Staubli VAL3: Cognex.dtx

bool bCheckRowUpLim = true
bool bDebugProgram = true
bool bDebugSocket
bool bGetID
bool bSafe
bool l_bError
bool resultTrigger = true
camera cCamera[11]
  [0]
    num nErrorCode = 70
    string sErrorMsg[121]
      [0] = "Login> Unrecognized command"
      [1] = "Login> Wrong user name or password"
      [2] = "Login> Communication Error"
      [10] = "Set Online> Command successfull"
      [11] = "Set Online> Unrecognized command"
      [12] = "Set Online> The value given for Int is either out of range, or is not a valid integer"
      [13] = "Set Online> The command could not be executed"
      [14] = "Set Online> Sensor is set Offline manually "
      [15] = "Set Online> User does not have Full Access to execute the command."
      [20] = "Get Online> The In-Sight sensor is currently Offline"
      [21] = "Get Online> The In-Sight sensor is currently Online"
      [30] = "Load File> Command successfull"
      [31] = "Load File> Unrecognized command"
      [32] = "Load File> The filename is missing"
      [33] = "Load File> The job failed to load, the sensor is Online, or the file was not found"
      [34] = "Load File> The job to be loaded was not found, or the sensor is out of memory"
      [35] = "Load File> User does not have Full Access"
      [40] = "get File> Command successfull"
      [41] = "get File> Unrecognized command"
      [42] = "get File> The active job has not been saved"
      [50] = "Save file> Command successfull"
      [51] = "Save file> Unrecognized command"
      [52] = "Save file> The filename is missing"
      [53] = "Save file>The job failed to save, the sensor is Online or the file was not found"
      [54] = "Save file> User does not have Full Access "
      [60] = "Set Event> Command successfull"
      [61] = "Set Event> Unrecognized command"
      [62] = "Set Event> The number is either out of range or not an integer"
      [63] = "Set Event>The command could not be executed, or the sensor is Offline"
      [64] = "Set Event> User does not have Full Access "
      [70] = "Get Value> Command successfull"
      [71] = "Get Value> Unrecognized command"
      [72] = "Get Value> Cell ID is invalid"
      [73] = "Get Value> The command could not be executed"
      [80] = "Set Float> Command successfull"
      [81] = "Set Float> Unrecognized command"
      [82] = "Set Float> Cell ID is invalid, or not a float"
      [83] = "Set Float> Cell was not created by the EditFloat function"
      [84] = "Set Float> User does not have Full Access "
      [90] = "Set Integer> Command successfull"
      [91] = "Set Integer>Unrecognized command"
      [92] = "Set Integer>Cell ID invalid, or not an integer"
      [93] = "Set Integer> Integer value is outside of the control's valid range or cell was not created by the EditInt function"
      [94] = "Set Integer> User does not have Full Access"
      [100] = "Set String> Command successfull"
      [101] = "Set String> Unrecognized command"
      [102] = "Set String> Cell ID invalid"
      [103] = "Set String> String is too longer or the cell does not contain an EditString function"
      [104] = "Set String> User does not have Full Access"
      [110] = "Cell Format> OK"
      [111] = "Cell Format> Invalid column"
      [112] = "Cell Format> Invalid row"
      [113] = "Cell Format> Row number out of range"
    sio sSocket = {link=Socket\sCognex1}
    bool bConnected
  [1]
    num nErrorCode = 70
    string sErrorMsg[120]
      [0] = "Login> Unrecognized command"
      [1] = "Login> Wrong user name or password"
      [2] = "Login> Communication Error"
      [10] = "Set Online> Command successfully"
      [11] = "Set Online> Unrecognized command"
      [12] = "Set Online> The value given for Int is either out of range, or is not a valid integer"
      [13] = "Set Online> The command could not be executed"
      [14] = "Set Online> Sensor is set Offline manually "
      [15] = "Set Online> User does not have Full Access to execute the command."
      [20] = "Get Online> The In-Sight sensor is currently Offline"
      [21] = "Get Online> The In-Sight sensor is currently Online"
      [30] = "Load File> Command successfully"
      [31] = "Load File> Unrecognized command"
      [32] = "Load File> The filename is missing"
      [33] = "Load File> The job failed to load, the sensor is Online, or the file was not found"
      [34] = "Load File> The job to be loaded was not found, or the sensor is out of memory"
      [35] = "Load File> User does not have Full Access"
      [40] = "get File> Command successfully"
      [41] = "get File> Unrecognized command"
      [42] = "get File> The active job has not been saved"
      [50] = "Save file> Command successfully"
      [51] = "Save file> Unrecognized command"
      [52] = "Save file> The filename is missing"
      [53] = "Save file>The job failed to save, the sensor is Online or the file was not found"
      [54] = "Save file> User does not have Full Access "
      [60] = "Set Event> Command successfully"
      [61] = "Set Event> Unrecognized command"
      [62] = "Set Event> The number is either out of range or not an integer"
      [63] = "Set Event>The command could not be executed, or the sensor is Offline"
      [64] = "Set Event> User does not have Full Access "
      [70] = "Get Value> Command successfully"
      [71] = "Get Value> Unrecognized command"
      [72] = "Get Value> Cell ID is invalid"
      [73] = "Get Value> The command could not be executed"
      [80] = "Set Float> Command successfully"
      [81] = "Set Float> Unrecognized command"
      [82] = "Set Float> Cell ID is invalid, or not a float"
      [83] = "Set Float> Cell was not created by the EditFloat function"
      [84] = "Set Float> User does not have Full Access "
      [90] = "Set Integer> Command successfully"
      [91] = "Set Integer>Unrecognized command"
      [92] = "Set Integer>Cell ID invalid, or not an integer"
      [93] = "Set Integer> Integer value is outside of the control's valid range or cell was not created by the EditInt function"
      [94] = "Set Integer> User does not have Full Access"
      [100] = "Set String> Command successfully"
      [101] = "Set String> Unrecognized command"
      [102] = "Set String> Cell ID invalid"
      [103] = "Set String> String is too longer or the cell does not contain an EditString function"
      [104] = "Set String> User does not have Full Access"
      [110] = "Cell Format> OK"
      [111] = "Cell Format> Invalid column"
      [112] = "Cell Format> Invalid row"
      [113] = "Cell Format> Row number out of range"
    sio sSocket = {link=Socket\sCognex1}
    bool bConnected
  [2]
    num nErrorCode
    string sErrorMsg[120]
      [0] = "Login> Unrecognized command"
      [1] = "Login> Wrong user name or password"
      [2] = "Login> Communication Error"
      [10] = "Set Online> Command successfully"
      [11] = "Set Online> Unrecognized command"
      [12] = "Set Online> The value given for Int is either out of range, or is not a valid integer"
      [13] = "Set Online> The command could not be executed"
      [14] = "Set Online> Sensor is set Offline manually "
      [15] = "Set Online> User does not have Full Access to execute the command."
      [20] = "Get Online> The In-Sight sensor is currently Offline"
      [21] = "Get Online> The In-Sight sensor is currently Online"
      [30] = "Load File> Command successfully"
      [31] = "Load File> Unrecognized command"
      [32] = "Load File> The filename is missing"
      [33] = "Load File> The job failed to load, the sensor is Online, or the file was not found"
      [34] = "Load File> The job to be loaded was not found, or the sensor is out of memory"
      [35] = "Load File> User does not have Full Access"
      [40] = "get File> Command successfully"
      [41] = "get File> Unrecognized command"
      [42] = "get File> The active job has not been saved"
      [50] = "Save file> Command successfully"
      [51] = "Save file> Unrecognized command"
      [52] = "Save file> The filename is missing"
      [53] = "Save file>The job failed to save, the sensor is Online or the file was not found"
      [54] = "Save file> User does not have Full Access "
      [60] = "Set Event> Command successfully"
      [61] = "Set Event> Unrecognized command"
      [62] = "Set Event> The number is either out of range or not an integer"
      [63] = "Set Event>The command could not be executed, or the sensor is Offline"
      [64] = "Set Event> User does not have Full Access "
      [70] = "Get Value> Command successfully"
      [71] = "Get Value> Unrecognized command"
      [72] = "Get Value> Cell ID is invalid"
      [73] = "Get Value> The command could not be executed"
      [80] = "Set Float> Command successfully"
      [81] = "Set Float> Unrecognized command"
      [82] = "Set Float> Cell ID is invalid, or not a float"
      [83] = "Set Float> Cell was not created by the EditFloat function"
      [84] = "Set Float> User does not have Full Access "
      [90] = "Set Integer> Command successfully"
      [91] = "Set Integer>Unrecognized command"
      [92] = "Set Integer>Cell ID invalid, or not an integer"
      [93] = "Set Integer> Integer value is outside of the control's valid range or cell was not created by the EditInt function"
      [94] = "Set Integer> User does not have Full Access"
      [100] = "Set String> Command successfully"
      [101] = "Set String> Unrecognized command"
      [102] = "Set String> Cell ID invalid"
      [103] = "Set String> String is too longer or the cell does not contain an EditString function"
      [104] = "Set String> User does not have Full Access"
      [110] = "Cell Format> OK"
      [111] = "Cell Format> Invalid column"
      [112] = "Cell Format> Invalid row"
      [113] = "Cell Format> Row number out of range"
    sio sSocket
    bool bConnected
  [3]
    num nErrorCode
    string sErrorMsg[120]
      [0] = "Login> Unrecognized command"
      [1] = "Login> Wrong user name or password"
      [2] = "Login> Communication Error"
      [10] = "Set Online> Command successfully"
      [11] = "Set Online> Unrecognized command"
      [12] = "Set Online> The value given for Int is either out of range, or is not a valid integer"
      [13] = "Set Online> The command could not be executed"
      [14] = "Set Online> Sensor is set Offline manually "
      [15] = "Set Online> User does not have Full Access to execute the command."
      [20] = "Get Online> The In-Sight sensor is currently Offline"
      [21] = "Get Online> The In-Sight sensor is currently Online"
      [30] = "Load File> Command successfully"
      [31] = "Load File> Unrecognized command"
      [32] = "Load File> The filename is missing"
      [33] = "Load File> The job failed to load, the sensor is Online, or the file was not found"
      [34] = "Load File> The job to be loaded was not found, or the sensor is out of memory"
      [35] = "Load File> User does not have Full Access"
      [40] = "get File> Command successfully"
      [41] = "get File> Unrecognized command"
      [42] = "get File> The active job has not been saved"
      [50] = "Save file> Command successfully"
      [51] = "Save file> Unrecognized command"
      [52] = "Save file> The filename is missing"
      [53] = "Save file>The job failed to save, the sensor is Online or the file was not found"
      [54] = "Save file> User does not have Full Access "
      [60] = "Set Event> Command successfully"
      [61] = "Set Event> Unrecognized command"
      [62] = "Set Event> The number is either out of range or not an integer"
      [63] = "Set Event>The command could not be executed, or the sensor is Offline"
      [64] = "Set Event> User does not have Full Access "
      [70] = "Get Value> Command successfully"
      [71] = "Get Value> Unrecognized command"
      [72] = "Get Value> Cell ID is invalid"
      [73] = "Get Value> The command could not be executed"
      [80] = "Set Float> Command successfully"
      [81] = "Set Float> Unrecognized command"
      [82] = "Set Float> Cell ID is invalid, or not a float"
      [83] = "Set Float> Cell was not created by the EditFloat function"
      [84] = "Set Float> User does not have Full Access "
      [90] = "Set Integer> Command successfully"
      [91] = "Set Integer>Unrecognized command"
      [92] = "Set Integer>Cell ID invalid, or not an integer"
      [93] = "Set Integer> Integer value is outside of the control's valid range or cell was not created by the EditInt function"
      [94] = "Set Integer> User does not have Full Access"
      [100] = "Set String> Command successfully"
      [101] = "Set String> Unrecognized command"
      [102] = "Set String> Cell ID invalid"
      [103] = "Set String> String is too longer or the cell does not contain an EditString function"
      [104] = "Set String> User does not have Full Access"
      [110] = "Cell Format> OK"
      [111] = "Cell Format> Invalid column"
      [112] = "Cell Format> Invalid row"
      [113] = "Cell Format> Row number out of range"
    sio sSocket
    bool bConnected
  [4]
    num nErrorCode
    string sErrorMsg[120]
      [0] = "Login> Unrecognized command"
      [1] = "Login> Wrong user name or password"
      [2] = "Login> Communication Error"
      [10] = "Set Online> Command successfully"
      [11] = "Set Online> Unrecognized command"
      [12] = "Set Online> The value given for Int is either out of range, or is not a valid integer"
      [13] = "Set Online> The command could not be executed"
      [14] = "Set Online> Sensor is set Offline manually "
      [15] = "Set Online> User does not have Full Access to execute the command."
      [20] = "Get Online> The In-Sight sensor is currently Offline"
      [21] = "Get Online> The In-Sight sensor is currently Online"
      [30] = "Load File> Command successfully"
      [31] = "Load File> Unrecognized command"
      [32] = "Load File> The filename is missing"
      [33] = "Load File> The job failed to load, the sensor is Online, or the file was not found"
      [34] = "Load File> The job to be loaded was not found, or the sensor is out of memory"
      [35] = "Load File> User does not have Full Access"
      [40] = "get File> Command successfully"
      [41] = "get File> Unrecognized command"
      [42] = "get File> The active job has not been saved"
      [50] = "Save file> Command successfully"
      [51] = "Save file> Unrecognized command"
      [52] = "Save file> The filename is missing"
      [53] = "Save file>The job failed to save, the sensor is Online or the file was not found"
      [54] = "Save file> User does not have Full Access "
      [60] = "Set Event> Command successfully"
      [61] = "Set Event> Unrecognized command"
      [62] = "Set Event> The number is either out of range or not an integer"
      [63] = "Set Event>The command could not be executed, or the sensor is Offline"
      [64] = "Set Event> User does not have Full Access "
      [70] = "Get Value> Command successfully"
      [71] = "Get Value> Unrecognized command"
      [72] = "Get Value> Cell ID is invalid"
      [73] = "Get Value> The command could not be executed"
      [80] = "Set Float> Command successfully"
      [81] = "Set Float> Unrecognized command"
      [82] = "Set Float> Cell ID is invalid, or not a float"
      [83] = "Set Float> Cell was not created by the EditFloat function"
      [84] = "Set Float> User does not have Full Access "
      [90] = "Set Integer> Command successfully"
      [91] = "Set Integer>Unrecognized command"
      [92] = "Set Integer>Cell ID invalid, or not an integer"
      [93] = "Set Integer> Integer value is outside of the control's valid range or cell was not created by the EditInt function"
      [94] = "Set Integer> User does not have Full Access"
      [100] = "Set String> Command successfully"
      [101] = "Set String> Unrecognized command"
      [102] = "Set String> Cell ID invalid"
      [103] = "Set String> String is too longer or the cell does not contain an EditString function"
      [104] = "Set String> User does not have Full Access"
      [110] = "Cell Format> OK"
      [111] = "Cell Format> Invalid column"
      [112] = "Cell Format> Invalid row"
      [113] = "Cell Format> Row number out of range"
    sio sSocket
    bool bConnected
  [5]
    num nErrorCode
    string sErrorMsg[120]
      [0] = "Login> Unrecognized command"
      [1] = "Login> Wrong user name or password"
      [2] = "Login> Communication Error"
      [10] = "Set Online> Command successfully"
      [11] = "Set Online> Unrecognized command"
      [12] = "Set Online> The value given for Int is either out of range, or is not a valid integer"
      [13] = "Set Online> The command could not be executed"
      [14] = "Set Online> Sensor is set Offline manually "
      [15] = "Set Online> User does not have Full Access to execute the command."
      [20] = "Get Online> The In-Sight sensor is currently Offline"
      [21] = "Get Online> The In-Sight sensor is currently Online"
      [30] = "Load File> Command successfully"
      [31] = "Load File> Unrecognized command"
      [32] = "Load File> The filename is missing"
      [33] = "Load File> The job failed to load, the sensor is Online, or the file was not found"
      [34] = "Load File> The job to be loaded was not found, or the sensor is out of memory"
      [35] = "Load File> User does not have Full Access"
      [40] = "get File> Command successfully"
      [41] = "get File> Unrecognized command"
      [42] = "get File> The active job has not been saved"
      [50] = "Save file> Command successfully"
      [51] = "Save file> Unrecognized command"
      [52] = "Save file> The filename is missing"
      [53] = "Save file>The job failed to save, the sensor is Online or the file was not found"
      [54] = "Save file> User does not have Full Access "
      [60] = "Set Event> Command successfully"
      [61] = "Set Event> Unrecognized command"
      [62] = "Set Event> The number is either out of range or not an integer"
      [63] = "Set Event>The command could not be executed, or the sensor is Offline"
      [64] = "Set Event> User does not have Full Access "
      [70] = "Get Value> Command successfully"
      [71] = "Get Value> Unrecognized command"
      [72] = "Get Value> Cell ID is invalid"
      [73] = "Get Value> The command could not be executed"
      [80] = "Set Float> Command successfully"
      [81] = "Set Float> Unrecognized command"
      [82] = "Set Float> Cell ID is invalid, or not a float"
      [83] = "Set Float> Cell was not created by the EditFloat function"
      [84] = "Set Float> User does not have Full Access "
      [90] = "Set Integer> Command successfully"
      [91] = "Set Integer>Unrecognized command"
      [92] = "Set Integer>Cell ID invalid, or not an integer"
      [93] = "Set Integer> Integer value is outside of the control's valid range or cell was not created by the EditInt function"
      [94] = "Set Integer> User does not have Full Access"
      [100] = "Set String> Command successfully"
      [101] = "Set String> Unrecognized command"
      [102] = "Set String> Cell ID invalid"
      [103] = "Set String> String is too longer or the cell does not contain an EditString function"
      [104] = "Set String> User does not have Full Access"
      [110] = "Cell Format> OK"
      [111] = "Cell Format> Invalid column"
      [112] = "Cell Format> Invalid row"
      [113] = "Cell Format> Row number out of range"
    sio sSocket
    bool bConnected
  [6]
    num nErrorCode
    string sErrorMsg[120]
      [0] = "Login> Unrecognized command"
      [1] = "Login> Wrong user name or password"
      [2] = "Login> Communication Error"
      [10] = "Set Online> Command successfully"
      [11] = "Set Online> Unrecognized command"
      [12] = "Set Online> The value given for Int is either out of range, or is not a valid integer"
      [13] = "Set Online> The command could not be executed"
      [14] = "Set Online> Sensor is set Offline manually "
      [15] = "Set Online> User does not have Full Access to execute the command."
      [20] = "Get Online> The In-Sight sensor is currently Offline"
      [21] = "Get Online> The In-Sight sensor is currently Online"
      [30] = "Load File> Command successfully"
      [31] = "Load File> Unrecognized command"
      [32] = "Load File> The filename is missing"
      [33] = "Load File> The job failed to load, the sensor is Online, or the file was not found"
      [34] = "Load File> The job to be loaded was not found, or the sensor is out of memory"
      [35] = "Load File> User does not have Full Access"
      [40] = "get File> Command successfully"
      [41] = "get File> Unrecognized command"
      [42] = "get File> The active job has not been saved"
      [50] = "Save file> Command successfully"
      [51] = "Save file> Unrecognized command"
      [52] = "Save file> The filename is missing"
      [53] = "Save file>The job failed to save, the sensor is Online or the file was not found"
      [54] = "Save file> User does not have Full Access "
      [60] = "Set Event> Command successfully"
      [61] = "Set Event> Unrecognized command"
      [62] = "Set Event> The number is either out of range or not an integer"
      [63] = "Set Event>The command could not be executed, or the sensor is Offline"
      [64] = "Set Event> User does not have Full Access "
      [70] = "Get Value> Command successfully"
      [71] = "Get Value> Unrecognized command"
      [72] = "Get Value> Cell ID is invalid"
      [73] = "Get Value> The command could not be executed"
      [80] = "Set Float> Command successfully"
      [81] = "Set Float> Unrecognized command"
      [82] = "Set Float> Cell ID is invalid, or not a float"
      [83] = "Set Float> Cell was not created by the EditFloat function"
      [84] = "Set Float> User does not have Full Access "
      [90] = "Set Integer> Command successfully"
      [91] = "Set Integer>Unrecognized command"
      [92] = "Set Integer>Cell ID invalid, or not an integer"
      [93] = "Set Integer> Integer value is outside of the control's valid range or cell was not created by the EditInt function"
      [94] = "Set Integer> User does not have Full Access"
      [100] = "Set String> Command successfully"
      [101] = "Set String> Unrecognized command"
      [102] = "Set String> Cell ID invalid"
      [103] = "Set String> String is too longer or the cell does not contain an EditString function"
      [104] = "Set String> User does not have Full Access"
      [110] = "Cell Format> OK"
      [111] = "Cell Format> Invalid column"
      [112] = "Cell Format> Invalid row"
      [113] = "Cell Format> Row number out of range"
    sio sSocket
    bool bConnected
  [7]
    num nErrorCode
    string sErrorMsg[120]
      [0] = "Login> Unrecognized command"
      [1] = "Login> Wrong user name or password"
      [2] = "Login> Communication Error"
      [10] = "Set Online> Command successfully"
      [11] = "Set Online> Unrecognized command"
      [12] = "Set Online> The value given for Int is either out of range, or is not a valid integer"
      [13] = "Set Online> The command could not be executed"
      [14] = "Set Online> Sensor is set Offline manually "
      [15] = "Set Online> User does not have Full Access to execute the command."
      [20] = "Get Online> The In-Sight sensor is currently Offline"
      [21] = "Get Online> The In-Sight sensor is currently Online"
      [30] = "Load File> Command successfully"
      [31] = "Load File> Unrecognized command"
      [32] = "Load File> The filename is missing"
      [33] = "Load File> The job failed to load, the sensor is Online, or the file was not found"
      [34] = "Load File> The job to be loaded was not found, or the sensor is out of memory"
      [35] = "Load File> User does not have Full Access"
      [40] = "get File> Command successfully"
      [41] = "get File> Unrecognized command"
      [42] = "get File> The active job has not been saved"
      [50] = "Save file> Command successfully"
      [51] = "Save file> Unrecognized command"
      [52] = "Save file> The filename is missing"
      [53] = "Save file>The job failed to save, the sensor is Online or the file was not found"
      [54] = "Save file> User does not have Full Access "
      [60] = "Set Event> Command successfully"
      [61] = "Set Event> Unrecognized command"
      [62] = "Set Event> The number is either out of range or not an integer"
      [63] = "Set Event>The command could not be executed, or the sensor is Offline"
      [64] = "Set Event> User does not have Full Access "
      [70] = "Get Value> Command successfully"
      [71] = "Get Value> Unrecognized command"
      [72] = "Get Value> Cell ID is invalid"
      [73] = "Get Value> The command could not be executed"
      [80] = "Set Float> Command successfully"
      [81] = "Set Float> Unrecognized command"
      [82] = "Set Float> Cell ID is invalid, or not a float"
      [83] = "Set Float> Cell was not created by the EditFloat function"
      [84] = "Set Float> User does not have Full Access "
      [90] = "Set Integer> Command successfully"
      [91] = "Set Integer>Unrecognized command"
      [92] = "Set Integer>Cell ID invalid, or not an integer"
      [93] = "Set Integer> Integer value is outside of the control's valid range or cell was not created by the EditInt function"
      [94] = "Set Integer> User does not have Full Access"
      [100] = "Set String> Command successfully"
      [101] = "Set String> Unrecognized command"
      [102] = "Set String> Cell ID invalid"
      [103] = "Set String> String is too longer or the cell does not contain an EditString function"
      [104] = "Set String> User does not have Full Access"
      [110] = "Cell Format> OK"
      [111] = "Cell Format> Invalid column"
      [112] = "Cell Format> Invalid row"
      [113] = "Cell Format> Row number out of range"
    sio sSocket
    bool bConnected
  [8]
    num nErrorCode
    string sErrorMsg[120]
      [0] = "Login> Unrecognized command"
      [1] = "Login> Wrong user name or password"
      [2] = "Login> Communication Error"
      [10] = "Set Online> Command successfully"
      [11] = "Set Online> Unrecognized command"
      [12] = "Set Online> The value given for Int is either out of range, or is not a valid integer"
      [13] = "Set Online> The command could not be executed"
      [14] = "Set Online> Sensor is set Offline manually "
      [15] = "Set Online> User does not have Full Access to execute the command."
      [20] = "Get Online> The In-Sight sensor is currently Offline"
      [21] = "Get Online> The In-Sight sensor is currently Online"
      [30] = "Load File> Command successfully"
      [31] = "Load File> Unrecognized command"
      [32] = "Load File> The filename is missing"
      [33] = "Load File> The job failed to load, the sensor is Online, or the file was not found"
      [34] = "Load File> The job to be loaded was not found, or the sensor is out of memory"
      [35] = "Load File> User does not have Full Access"
      [40] = "get File> Command successfully"
      [41] = "get File> Unrecognized command"
      [42] = "get File> The active job has not been saved"
      [50] = "Save file> Command successfully"
      [51] = "Save file> Unrecognized command"
      [52] = "Save file> The filename is missing"
      [53] = "Save file>The job failed to save, the sensor is Online or the file was not found"
      [54] = "Save file> User does not have Full Access "
      [60] = "Set Event> Command successfully"
      [61] = "Set Event> Unrecognized command"
      [62] = "Set Event> The number is either out of range or not an integer"
      [63] = "Set Event>The command could not be executed, or the sensor is Offline"
      [64] = "Set Event> User does not have Full Access "
      [70] = "Get Value> Command successfully"
      [71] = "Get Value> Unrecognized command"
      [72] = "Get Value> Cell ID is invalid"
      [73] = "Get Value> The command could not be executed"
      [80] = "Set Float> Command successfully"
      [81] = "Set Float> Unrecognized command"
      [82] = "Set Float> Cell ID is invalid, or not a float"
      [83] = "Set Float> Cell was not created by the EditFloat function"
      [84] = "Set Float> User does not have Full Access "
      [90] = "Set Integer> Command successfully"
      [91] = "Set Integer>Unrecognized command"
      [92] = "Set Integer>Cell ID invalid, or not an integer"
      [93] = "Set Integer> Integer value is outside of the control's valid range or cell was not created by the EditInt function"
      [94] = "Set Integer> User does not have Full Access"
      [100] = "Set String> Command successfully"
      [101] = "Set String> Unrecognized command"
      [102] = "Set String> Cell ID invalid"
      [103] = "Set String> String is too longer or the cell does not contain an EditString function"
      [104] = "Set String> User does not have Full Access"
      [110] = "Cell Format> OK"
      [111] = "Cell Format> Invalid column"
      [112] = "Cell Format> Invalid row"
      [113] = "Cell Format> Row number out of range"
    sio sSocket
    bool bConnected
  [9]
    num nErrorCode
    string sErrorMsg[120]
      [0] = "Login> Unrecognized command"
      [1] = "Login> Wrong user name or password"
      [2] = "Login> Communication Error"
      [10] = "Set Online> Command successfully"
      [11] = "Set Online> Unrecognized command"
      [12] = "Set Online> The value given for Int is either out of range, or is not a valid integer"
      [13] = "Set Online> The command could not be executed"
      [14] = "Set Online> Sensor is set Offline manually "
      [15] = "Set Online> User does not have Full Access to execute the command."
      [20] = "Get Online> The In-Sight sensor is currently Offline"
      [21] = "Get Online> The In-Sight sensor is currently Online"
      [30] = "Load File> Command successfully"
      [31] = "Load File> Unrecognized command"
      [32] = "Load File> The filename is missing"
      [33] = "Load File> The job failed to load, the sensor is Online, or the file was not found"
      [34] = "Load File> The job to be loaded was not found, or the sensor is out of memory"
      [35] = "Load File> User does not have Full Access"
      [40] = "get File> Command successfully"
      [41] = "get File> Unrecognized command"
      [42] = "get File> The active job has not been saved"
      [50] = "Save file> Command successfully"
      [51] = "Save file> Unrecognized command"
      [52] = "Save file> The filename is missing"
      [53] = "Save file>The job failed to save, the sensor is Online or the file was not found"
      [54] = "Save file> User does not have Full Access "
      [60] = "Set Event> Command successfully"
      [61] = "Set Event> Unrecognized command"
      [62] = "Set Event> The number is either out of range or not an integer"
      [63] = "Set Event>The command could not be executed, or the sensor is Offline"
      [64] = "Set Event> User does not have Full Access "
      [70] = "Get Value> Command successfully"
      [71] = "Get Value> Unrecognized command"
      [72] = "Get Value> Cell ID is invalid"
      [73] = "Get Value> The command could not be executed"
      [80] = "Set Float> Command successfully"
      [81] = "Set Float> Unrecognized command"
      [82] = "Set Float> Cell ID is invalid, or not a float"
      [83] = "Set Float> Cell was not created by the EditFloat function"
      [84] = "Set Float> User does not have Full Access "
      [90] = "Set Integer> Command successfully"
      [91] = "Set Integer>Unrecognized command"
      [92] = "Set Integer>Cell ID invalid, or not an integer"
      [93] = "Set Integer> Integer value is outside of the control's valid range or cell was not created by the EditInt function"
      [94] = "Set Integer> User does not have Full Access"
      [100] = "Set String> Command successfully"
      [101] = "Set String> Unrecognized command"
      [102] = "Set String> Cell ID invalid"
      [103] = "Set String> String is too longer or the cell does not contain an EditString function"
      [104] = "Set String> User does not have Full Access"
      [110] = "Cell Format> OK"
      [111] = "Cell Format> Invalid column"
      [112] = "Cell Format> Invalid row"
      [113] = "Cell Format> Row number out of range"
    sio sSocket
    bool bConnected
  [10]
    num nErrorCode
    string sErrorMsg[121]
      [0] = "Login> Unrecognized command"
      [1] = "Login> Wrong user name or password"
      [2] = "Login> Communication Error"
      [10] = "Set Online> Command successfully"
      [11] = "Set Online> Unrecognized command"
      [12] = "Set Online> The value given for Int is either out of range, or is not a valid integer"
      [13] = "Set Online> The command could not be executed"
      [14] = "Set Online> Sensor is set Offline manually "
      [15] = "Set Online> User does not have Full Access to execute the command."
      [20] = "Get Online> The In-Sight sensor is currently Offline"
      [21] = "Get Online> The In-Sight sensor is currently Online"
      [30] = "Load File> Command successfully"
      [31] = "Load File> Unrecognized command"
      [32] = "Load File> The filename is missing"
      [33] = "Load File> The job failed to load, the sensor is Online, or the file was not found"
      [34] = "Load File> The job to be loaded was not found, or the sensor is out of memory"
      [35] = "Load File> User does not have Full Access"
      [40] = "get File> Command successfully"
      [41] = "get File> Unrecognized command"
      [42] = "get File> The active job has not been saved"
      [50] = "Save file> Command successfully"
      [51] = "Save file> Unrecognized command"
      [52] = "Save file> The filename is missing"
      [53] = "Save file>The job failed to save, the sensor is Online or the file was not found"
      [54] = "Save file> User does not have Full Access "
      [60] = "Set Event> Command successfully"
      [61] = "Set Event> Unrecognized command"
      [62] = "Set Event> The number is either out of range or not an integer"
      [63] = "Set Event>The command could not be executed, or the sensor is Offline"
      [64] = "Set Event> User does not have Full Access "
      [70] = "Get Value> Command successfully"
      [71] = "Get Value> Unrecognized command"
      [72] = "Get Value> Cell ID is invalid"
      [73] = "Get Value> The command could not be executed"
      [80] = "Set Float> Command successfully"
      [81] = "Set Float> Unrecognized command"
      [82] = "Set Float> Cell ID is invalid, or not a float"
      [83] = "Set Float> Cell was not created by the EditFloat function"
      [84] = "Set Float> User does not have Full Access "
      [90] = "Set Integer> Command successfully"
      [91] = "Set Integer>Unrecognized command"
      [92] = "Set Integer>Cell ID invalid, or not an integer"
      [93] = "Set Integer> Integer value is outside of the control's valid range or cell was not created by the EditInt function"
      [94] = "Set Integer> User does not have Full Access"
      [100] = "Set String> Command successfully"
      [101] = "Set String> Unrecognized command"
      [102] = "Set String> Cell ID invalid"
      [103] = "Set String> String is too longer or the cell does not contain an EditString function"
      [104] = "Set String> User does not have Full Access"
      [110] = "Cell Format> OK"
      [111] = "Cell Format> Invalid column"
      [112] = "Cell Format> Invalid row"
      [113] = "Cell Format> Row number out of range"
    sio sSocket
    bool bConnected
dio bbleu = {link=BasicIO-1\%I6}
dio borange = {link=BasicIO-1\%I1}
dio brouge = {link=BasicIO-1\%I2}
dio bvert = {link=BasicIO-1\%I3}
dio safe3 = {link=BasicIO-1\%Q4}
dio vbleu = {link=BasicIO-1\%Q0}
dio vorange = {link=BasicIO-1\%Q1}
dio vrouge = {link=BasicIO-1\%Q2}
dio vvert = {link=BasicIO-1\%Q3}
frame fcamera = {x=-304.013827, y=-243.818264, z=-221.906385, rx=-0.002067, ry=-0.000266, rz=-92.308469, fatherId=world[0]}
mdesc lent = {accel=2.25, vel=15, decel=2.25}
mdesc rapide
num nCamID
num nLibErrorCode
num nProgram[10]
  [0] = 8
  [1] = 1
num nbPoint
num resultx = -4.409
num resulty = 7.256
num resultz = 3.056
pointRx AxeX = {x=-305.715465, y=-286.02975, z=-221.90487, rx=-0.188763, ry=179.501609, rz=-1.345575, fatherId=world[0]}
pointRx AxeY = {x=-257.758895, y=-245.465285, z=-221.906111, rx=-0.187758, ry=179.500593, rz=-1.345622, fatherId=world[0]}
pointRx Origine = {x=-304.013827, y=-243.818264, z=-221.906385, rx=-0.188173, ry=179.50125, rz=-1.345489, fatherId=world[0]}
pointRx PointCamera = {x=-4.409, y=7.256, z=55.5, rx=180, rz=90, fatherId=fcamera[0]}
pointRx PointDePassage = {x=46.369415, y=-346.332649, z=138.873975, rx=0.118221, ry=178.943897, rz=-76.444907, fatherId=world[0]}
pointRx PointDePause = {fatherId=world[0]}
pointRx PointDePose = {x=431.860377, y=24.045354, z=-29.900035, rx=-179.634859, ry=0.400912, rz=18.010944, fatherId=world[0]}
pointRx PointDePoseHaut = {x=431.86073, y=24.045369, z=65.602019, rx=-179.63482, ry=0.401543, rz=18.010937, fatherId=world[0]}
sio sCognex = {link=Socket\sCognex1}
string Prisephoto
string result
string sLibError[300]
  [200] = "isIDAvailable> ID not available"
  [201] = "getNextID> No more IDs available"
  [202] = "checkErrFormat> Not logged into camera"
  [203] = "login> ID not available (already tied to a camera)"
string strVersion = "7.3.1.0"
tool pince = {fatherId=flange[0], ioLink=valve1}
